// TIA Portal project "Automated_Pumping_Station" (V17)

(* hardware
DEVICE "HMI_1"  TP700 Comfort
   slot 0: "HMI_1"  TP700 Comfort  6AV2 124-0GC01-0AX0  17.0.0.0
   slot 1: "HMI_RT_1"  TP700 Comfort  6AV2 124-0GC01-0AX0  17.0.0.0
   slot 5: "HMI_1.IE_CP_1"  PROFINET Interface  17.0.0.0
      slot 1: "PROFINET Interface_1"  PROFINET Interface
         slot 1: "Port_1"  Port
         slot 2: "Port_2"  Port
   slot 7: "HMI_1.MPI/DP_CP_1"  MPI/DP Interface  17.0.0.0
DEVICE "S7-1500/ET200MP station_1"  S7-1500 station
   slot 0: "Rail_0"  Rack  6ES7 590-1***0-0AA0
   slot 1: "PLC_1"  CPU 1511-1 PN  6ES7 511-1AK00-0AB0  V1.8
      slot 3: "CPU display_1"  6ES7591-1AA00-0AA0
      slot 32768: "PROFINET interface_1"  X1
         slot 32769: "Port_1"  X1 P1
         slot 32770: "Port_2"  X1 P2
   slot 2: "DI 16x24VDC / DQ 16x24VDC/0.5A BA_1"  DI 16x24VDC/DQ 16x24VDC/0.5A BA  6ES7 523-1BL00-0AA0  V1.1
   slot 3: "AI 8xU/I HS_1"  AI 8xU/I HS  6ES7 531-7NF10-0AB0  V2.1
*)

// ===== PLC "PLC_1"  CPU 1511-1 PN =====

VAR_GLOBAL   // PLC tag table "Default tag table"
   "AI_Raw_Line_Pressure" AT %IW96 : Int;   // Raw 4-20mA current loop from pressure sensor PT-101.
   "DI_Suction_Valve_Open" AT %I2.0 : Bool;   // Limit switch ZS-101 confirming the main water supply valve is fully open.
   "Stop Button" AT %I2.1 : Bool;   // Auxiliary contactor bit from Pump 1 motor starter circuit.
   "DI_Pump2_Feedback" AT %I2.2 : Bool;   // Auxiliary contactor bit from Pump 2 motor starter circuit.
   "DQ_Pump1_Start" AT %Q2.0 : Bool;   // Triggers the magnetic contactor coil to run Pump Motor 1.
   "DQ_Pump2_Start" AT %Q2.1 : Bool;   // Triggers the magnetic contactor coil to run Pump Motor 2.
   "TMP_Normalized_Pressure" AT %MD20 : Real;
   "Tag_1" AT %QW30 : Int;
   "AI_Raw_Flow_Meter" AT %IW98 : Int;
   "Dry_Run_Fault" AT %M10.0 : Bool;
   "alarms.Reset_Button" AT %I2.3 : Bool;
   "Reset_Light" AT %Q0.1 : Bool;
   "Knob" AT %IW100 : Int;
   "Process_Values.Status_Pressure" AT %MD30 : Real;
   "SP_lcd" AT %QW34 : Int;
   "TMP_Normalized_SP" AT %MD35 : Real;
   "Ramp_Complete" AT %M40.0 : Bool;
   "Stop light" AT %Q0.2 : Bool;
   "System_Byte" AT %MB1 : Byte;
   "FirstScan" AT %M1.0 : Bool;
   "DiagStatusUpdate" AT %M1.1 : Bool;
   "AlwaysTRUE" AT %M1.2 : Bool;
   "AlwaysFALSE" AT %M1.3 : Bool;
   "Clock_Byte" AT %MB0 : Byte;
   "Clock_10Hz" AT %M0.0 : Bool;
   "Clock_5Hz" AT %M0.1 : Bool;
   "Clock_2.5Hz" AT %M0.2 : Bool;
   "Clock_2Hz" AT %M0.3 : Bool;
   "Clock_1.25Hz" AT %M0.4 : Bool;
   "Clock_1Hz" AT %M0.5 : Bool;
   "Clock_0.625Hz" AT %M0.6 : Bool;
   "Clock_0.5Hz" AT %M0.7 : Bool;
   "Manual_Ramp_Output" AT %MW50 : Int;
   "PID_Output_Value" AT %MW52 : Int;
   "Tag_2" AT %I0.3 : Bool;
   "PV" AT %QW36 : Int;
   "Level_Error" AT %MD60 : Real;
   "Raw_Math_Output" AT %MD64 : Real;
END_VAR

DATA_BLOCK "DB_HMI_Interface"   // DB1
{ S7_Optimized_Access := 'TRUE' }
VERSION : 0.1
   VAR
      Process_Values : Struct   // Collapsible structure to group all live plant readings.
         Status_Pressure : Real := 0.0;   // Calculated line pressure in Bar passed from SCALE_X.
      END_STRUCT;
      alarms : Struct
         High_Pressure_Fault : Bool;
         Reset_Button : Bool;
      END_STRUCT;
      Control_Commands : Struct   // Grouping for manual HMI operator commands.
         Pump1_Start_HMI : Bool;   // Momentary push-button from HMI to start Pump 1.
         Pump1_Stop_HMI : Bool;   // Momentary push-button from HMI to stop Pump 1.
      END_STRUCT;
   END_VAR
BEGIN
END_DATA_BLOCK

// folder: System blocks/Program resources

DATA_BLOCK "IEC_Timer_0_DB"   // DB2
{ S7_Optimized_Access := 'TRUE' }
AUTHOR : Simatic
FAMILY : IEC
NAME : IEC_TMR
VERSION : 1.0
// stored: InstanceOfName IEC_TIMER
"IEC_TIMER"
BEGIN
END_DATA_BLOCK

// folder: (top level)

ORGANIZATION_BLOCK "Main"   // OB1, LAD, ProgramCycle
TITLE = "Main Program Sweep (Cycle)"
{ S7_Optimized_Access := 'TRUE' }
VERSION : 0.1
   VAR_INPUT
      Initial_Call : Bool;   // Initial call of this OB
      Remanence : Bool;   // =True, if remanent data are available
   END_VAR
BEGIN

REGION Network 1
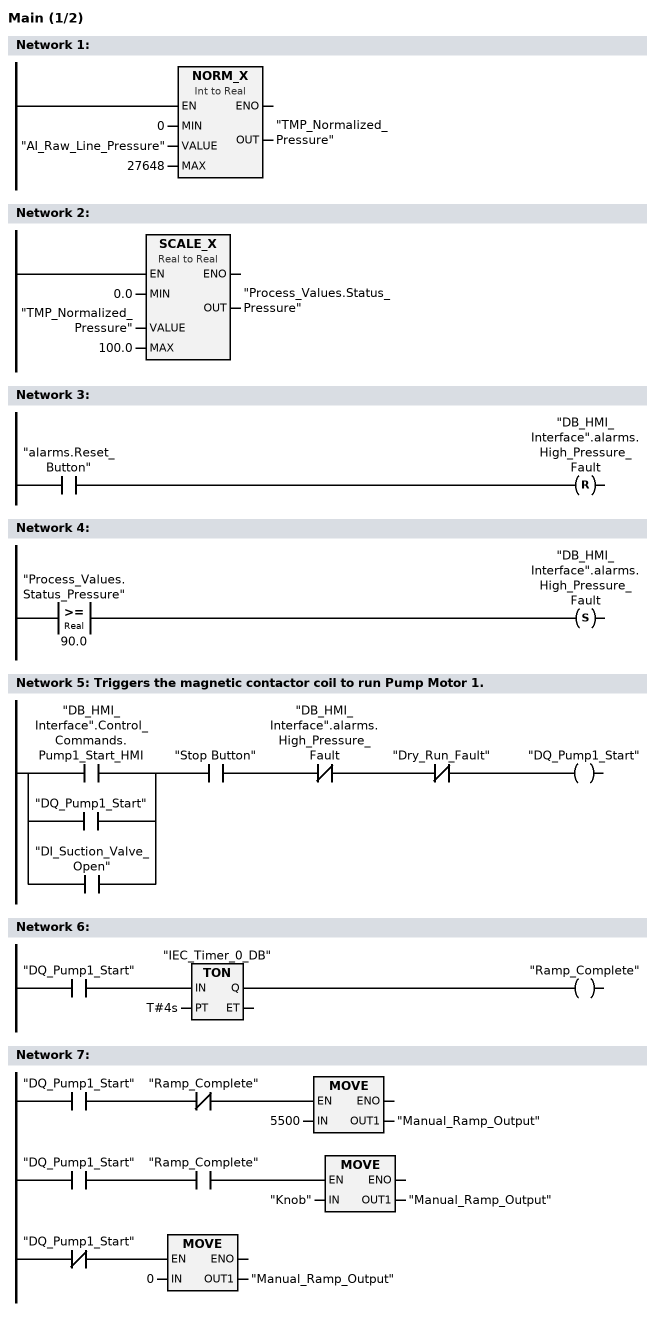
   RUNG wire#powerrail
      { S7_Templates := "[SrcType := Int, DestType := Real]" } Normalize(min := 0, value := "AI_Raw_Line_Pressure", max := 27648, out => "TMP_Normalized_Pressure")
   END_RUNG
   // the same network as SCL:
   "TMP_Normalized_Pressure" := NORM_X(MIN := 0, VALUE := "AI_Raw_Line_Pressure", MAX := 27648);
END_REGION

REGION Network 2
   RUNG wire#powerrail
      { S7_Templates := "[SrcType := Real, DestType := Real]" } Scale(min := 0.0, value := "TMP_Normalized_Pressure", max := 100.0, out => "Process_Values.Status_Pressure")
   END_RUNG
   // the same network as SCL:
   "Process_Values.Status_Pressure" := SCALE_X(MIN := 0.0, VALUE := "TMP_Normalized_Pressure", MAX := 100.0);
END_REGION

REGION Network 3
   RUNG wire#powerrail
      Contact( "alarms.Reset_Button" )
      R_Coil( "DB_HMI_Interface".alarms.High_Pressure_Fault )
   END_RUNG
   // the same network as SCL:
   IF "alarms.Reset_Button" THEN "DB_HMI_Interface".alarms.High_Pressure_Fault := FALSE; END_IF;
END_REGION

REGION Network 4
   RUNG wire#powerrail
      { S7_Templates := "SrcType := Real" } GE_Contact(in1 := "Process_Values.Status_Pressure", in2 := 90.0)
      S_Coil( "DB_HMI_Interface".alarms.High_Pressure_Fault )
   END_RUNG
   // the same network as SCL:
   IF "Process_Values.Status_Pressure" >= 90.0 THEN
       "DB_HMI_Interface".alarms.High_Pressure_Fault := TRUE;
   END_IF;
END_REGION

REGION Network 5: Triggers the magnetic contactor coil to run Pump Motor 1.
   RUNG wire#powerrail
      Contact( "DB_HMI_Interface".Control_Commands.Pump1_Start_HMI )
      wire#w1
      Contact( "Stop Button" )
      I_Contact( "DB_HMI_Interface".alarms.High_Pressure_Fault )
      I_Contact( "Dry_Run_Fault" )
      Coil( "DQ_Pump1_Start" )
   END_RUNG
   RUNG wire#powerrail
      Contact( "DQ_Pump1_Start" )
   END_RUNG wire#w1
   RUNG wire#powerrail
      Contact( "DI_Suction_Valve_Open" )
   END_RUNG wire#w1
   // the same network as SCL:
   "DQ_Pump1_Start" := ("DB_HMI_Interface".Control_Commands.Pump1_Start_HMI OR "DQ_Pump1_Start" OR "DI_Suction_Valve_Open") AND "Stop Button" AND NOT "DB_HMI_Interface".alarms.High_Pressure_Fault AND NOT "Dry_Run_Fault";
END_REGION

REGION Network 6
   "IEC_Timer_0_DB".TON(IN := "DQ_Pump1_Start", PT := T#4s);
   "Ramp_Complete" := "IEC_Timer_0_DB".Q;
END_REGION

REGION Network 7
   RUNG wire#powerrail
      Contact( "DQ_Pump1_Start" )
      I_Contact( "Ramp_Complete" )
      Move(in := 5500, out1 => "Manual_Ramp_Output")
   END_RUNG
   RUNG wire#powerrail
      Contact( "DQ_Pump1_Start" )
      Contact( "Ramp_Complete" )
      Move(in := "Knob", out1 => "Manual_Ramp_Output")
   END_RUNG
   RUNG wire#powerrail
      I_Contact( "DQ_Pump1_Start" )
      Move(in := 0, out1 => "Manual_Ramp_Output")
   END_RUNG
   // the same network as SCL:
   IF "DQ_Pump1_Start" AND NOT "Ramp_Complete" THEN "Manual_Ramp_Output" := 5500; END_IF;
   IF "DQ_Pump1_Start" AND "Ramp_Complete" THEN "Manual_Ramp_Output" := "Knob"; END_IF;
   IF NOT "DQ_Pump1_Start" THEN "Manual_Ramp_Output" := 0; END_IF;
END_REGION

REGION Network 8
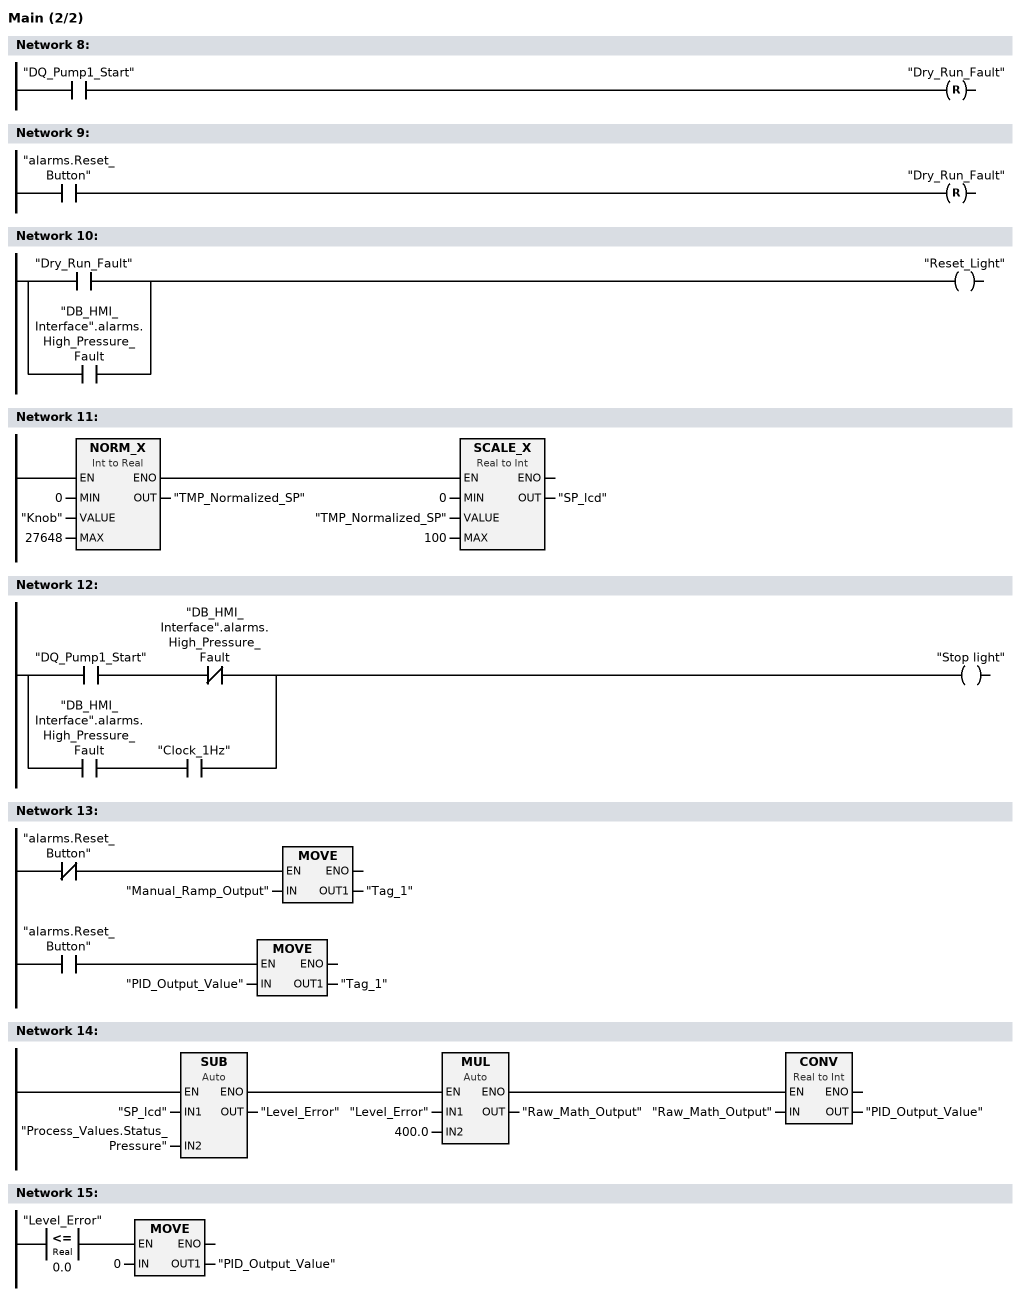
   RUNG wire#powerrail
      Contact( "DQ_Pump1_Start" )
      R_Coil( "Dry_Run_Fault" )
   END_RUNG
   // the same network as SCL:
   IF "DQ_Pump1_Start" THEN "Dry_Run_Fault" := FALSE; END_IF;
END_REGION

REGION Network 9
   RUNG wire#powerrail
      Contact( "alarms.Reset_Button" )
      R_Coil( "Dry_Run_Fault" )
   END_RUNG
   // the same network as SCL:
   IF "alarms.Reset_Button" THEN "Dry_Run_Fault" := FALSE; END_IF;
END_REGION

REGION Network 10
   RUNG wire#powerrail
      Contact( "Dry_Run_Fault" )
      wire#w1
      Coil( "Reset_Light" )
   END_RUNG
   RUNG wire#powerrail
      Contact( "DB_HMI_Interface".alarms.High_Pressure_Fault )
   END_RUNG wire#w1
   // the same network as SCL:
   "Reset_Light" := "Dry_Run_Fault" OR "DB_HMI_Interface".alarms.High_Pressure_Fault;
END_REGION

REGION Network 11
   RUNG wire#powerrail
      { S7_Templates := "[SrcType := Int, DestType := Real]" } Normalize(min := 0, value := "Knob", max := 27648, out => "TMP_Normalized_SP")
      { S7_Templates := "[SrcType := Real, DestType := Int]" } Scale(min := 0, value := "TMP_Normalized_SP", max := 100, out => "SP_lcd")
   END_RUNG
   // the same network as SCL:
   "TMP_Normalized_SP" := NORM_X(MIN := 0, VALUE := "Knob", MAX := 27648);
   "SP_lcd" := SCALE_X(MIN := 0, VALUE := "TMP_Normalized_SP", MAX := 100);
END_REGION

REGION Network 12
   RUNG wire#powerrail
      Contact( "DQ_Pump1_Start" )
      I_Contact( "DB_HMI_Interface".alarms.High_Pressure_Fault )
      wire#w1
      Coil( "Stop light" )
   END_RUNG
   RUNG wire#powerrail
      Contact( "DB_HMI_Interface".alarms.High_Pressure_Fault )
      Contact( "Clock_1Hz" )
   END_RUNG wire#w1
   // the same network as SCL:
   "Stop light" := ("DQ_Pump1_Start" AND NOT "DB_HMI_Interface".alarms.High_Pressure_Fault) OR ("DB_HMI_Interface".alarms.High_Pressure_Fault AND "Clock_1Hz");
END_REGION

REGION Network 13
   RUNG wire#powerrail
      I_Contact( "alarms.Reset_Button" )
      Move(in := "Manual_Ramp_Output", out1 => "Tag_1")
   END_RUNG
   RUNG wire#powerrail
      Contact( "alarms.Reset_Button" )
      Move(in := "PID_Output_Value", out1 => "Tag_1")
   END_RUNG
   // the same network as SCL:
   IF NOT "alarms.Reset_Button" THEN "Tag_1" := "Manual_Ramp_Output"; END_IF;
   IF "alarms.Reset_Button" THEN "Tag_1" := "PID_Output_Value"; END_IF;
END_REGION

REGION Network 14
   RUNG wire#powerrail
      Sub(in1 := "SP_lcd", in2 := "Process_Values.Status_Pressure", out => "Level_Error")
      Mul(in1 := "Level_Error", in2 := 400.0, out => "Raw_Math_Output")
      { S7_Templates := "[SrcType := Real, DestType := Int]" } Convert(in := "Raw_Math_Output", out => "PID_Output_Value")
   END_RUNG
   // the same network as SCL:
   "Level_Error" := "SP_lcd" - "Process_Values.Status_Pressure";
   "Raw_Math_Output" := "Level_Error" * 400.0;
   "PID_Output_Value" := REAL_TO_INT("Raw_Math_Output");
END_REGION

REGION Network 15
   RUNG wire#powerrail
      { S7_Templates := "SrcType := Real" } LE_Contact(in1 := "Level_Error", in2 := 0.0)
      Move(in := 0, out1 => "PID_Output_Value")
   END_RUNG
   // the same network as SCL:
   IF "Level_Error" <= 0.0 THEN "PID_Output_Value" := 0; END_IF;
END_REGION
END_ORGANIZATION_BLOCK

(* ===== HMI "HMI_RT_1" =====
system functions are stored by id; their names below are inferred from use

HMI tags "Default tag table"
   "Tag_ScreenNumber" : UInt, internal

screen "Root screen" 800x420, template "Template_1"
   on GenerateScreen: SetTag("Tag_ScreenNumber", 1)
   TextField "HmiScreenItemData" at 80,166 size 640x25; Text 'Welcome to HMI_1 (TP700 Comfort)!'

Template "Template_1" 800x420
   Button "Exit" at 720,360 size 78x58; TextOff 'Exit'; PictureOff "ExitRuntime_TP700_Comfort_TR"; PictureOn "ExitRuntime_TP700_Comfort_TR"
      on Release: StopRuntime(0)
   Button "Template_Button" at 640,360 size 78x58; TextOff 'Text'
   Button "Template_Button_1" at 560,360 size 78x58; TextOff 'Text'
   Button "Template_Button_2" at 480,360 size 78x58; TextOff 'Text'
   Button "Template_Button_3" at 400,360 size 78x58; TextOff 'Text'
   Button "Template_Button_4" at 321,360 size 78x58; TextOff 'Text'
   Button "Template_Button_5" at 241,360 size 78x58; TextOff 'Text'
   Button "Template_Button_6" at 161,360 size 78x58; TextOff 'Text'
   Button "Alarms" at 81,360 size 78x58; TextOff 'Alarms'; PictureOff "AlarmDisplay_TP700_Comfort_TR"; PictureOn "AlarmDisplay_TP700_Comfort_TR"
      on Release: function_ef3f5d25("Alarm window_Unacknowledged", -1)
   Button "Start screen" at 1,360 size 78x58; TextOff 'Start screen'; PictureOff "NavigateHome_TP700_Comfort_TR"; PictureOn "NavigateHome_TP700_Comfort_TR"
      on Release: ActivateScreen("Root screen", 0)
*)